(* CODESYS project SealBagSequence.xml

Project tree, tasks and I/O mapping:
  function block SealBagSequence [SFC]
*)

// SealBagSequence
FUNCTION_BLOCK SealBagSequence
// A function for stepping through bag sealing process.
// 
// When triggered this function will command the heat seal to close.
// Once confirmed closed, it will wait for the bag sealing delay
// time, and then open the heat seal. Once confirmed open it will pulse
// a completed bit.
//
// Any motion faults by the heat seal, failing to open or close in the 
// allowable time is managed by the heat seal motion sequence. This is
// a higher level function instructing the heat seal when to open and 
// close.
//  .					.					.
VAR_INPUT
	SFCInit: 			BOOL;				//
	Trigger: 			BOOL;				//
	HeatSealClosed: 	BOOL;				//
	HeatSealOpened: 	BOOL;				//
	SealingTime: 		TIME;				//
END_VAR
VAR_OUTPUT
	CloseHeatSeal: 		BOOL;				//
	OpenHeatSeal: 		BOOL;				//
	Complete: 			BOOL;				//
END_VAR
VAR
END_VAR

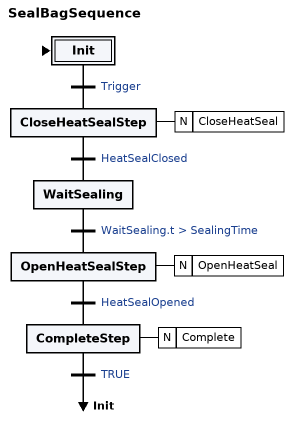
INITIAL_STEP Init:
END_STEP
TRANSITION FROM Init TO CloseHeatSealStep
    := Trigger;
END_TRANSITION
STEP CloseHeatSealStep:
    CloseHeatSeal(N);
END_STEP
TRANSITION FROM CloseHeatSealStep TO WaitSealing
    := HeatSealClosed;
END_TRANSITION
STEP WaitSealing:
END_STEP
TRANSITION FROM WaitSealing TO OpenHeatSealStep
    := WaitSealing.t > SealingTime;
END_TRANSITION
STEP OpenHeatSealStep:
    OpenHeatSeal(N);
END_STEP
TRANSITION FROM OpenHeatSealStep TO CompleteStep
    := HeatSealOpened;
END_TRANSITION
STEP CompleteStep:
    Complete(N);
END_STEP
TRANSITION FROM CompleteStep TO Init
    := TRUE;
END_TRANSITION

END_FUNCTION_BLOCK
